// Mitsubishi GX Works2 project: exercicio selo   PLC: Q03UDV

PROGRAM MAIN
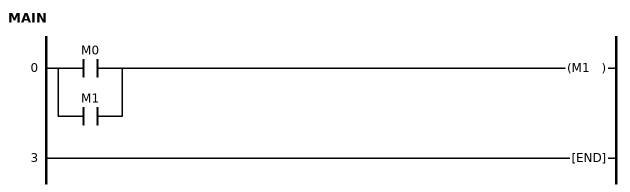
0     LD      M0
      OR      M1
      OUT     M1
3     END
END_PROGRAM
